{attribute 'qualified_only'}
{attribute 'strict'}
{attribute 'to_string'}
TYPE sStatesForTest :
(
	Target1Vektor := 0,
	CoordinatesInFrontOfTarget1,
	Wait1,
	Target1,
	Wait2,
	AfterTarget1,
	Target2Vector,
	CoordinatesInFrontOfTarget2,
	Wait3,
	Target2,
	Wait4,
	AfterTarget2,
	ParkingVector,
	Finished
);
END_TYPE

(* stored: Version 1.1.0.1, ProductVersion 3.1.4026.13
   DUT sStatesForTest: Id {f7ae5b27-5533-4627-879c-3ad1b5e00a44} *)
